(* IEC 61131-3 sources: plc_ladder_to_st/plc_export/st, 12 files *)

(* ---- P01_Main.st ---- *)
(* Generated ST from context: P01_Main *)
(* Project: plc project_260626 *)
(* CPU: QCPU (Q mode) Q06H *)

(* ============================================================ *)
(* [STEP 1] CODESYS > POU 열기 > DECLARATION(선언) 탭 > 아래만 붙여넣기 *)
(*          POU 이름과 PROGRAM 이름이 같아야 함: 'P01_Main' *)
(* ============================================================ *)

PROGRAM P01_Main
VAR
    SM400 : BOOL; (* 항상on *)
    M200 : BOOL; (* 제어전원ON *)
    X0 : BOOL; (* 운전준비ON [PBL] *)
    M201 : BOOL; (* 운전준비 PLS *)
    M202 : BOOL; (* 제어반 운전준비완료 *)
    M50 : BOOL; (* 제어반 비상정지 *)
    X1 : BOOL; (* 운전모드 자동[ ]  [SS] *)
    M210 : BOOL; (* 운전모드 수동[ ] *)
    M211 : BOOL; (* 운전모드 자동[ ] *)
    M500 : BOOL; (* 기동시작[HMI]   PB *)
    M215 : BOOL; (* 가와실러자동기동 *)
    M216 : BOOL; (* 현대 프라이머자동기동 *)
    M2127 : BOOL; (* 글라스 센터링 이상    TOTAL *)
    M2021 : BOOL; (* 글라스 센터링 운전준비 완료 *)
    X8 : BOOL; (* 이상해제[PB] *)
    M501 : BOOL; (* 이상해제[HMI]   PB *)
    M212 : BOOL; (* 이상해제 *)
    Y77 : BOOL; (* 선두 이더넷 카드 이상해제XY60 *)
    M502 : BOOL; (* 부저정지[HMI]   PB *)
    M220 : BOOL; (* 부져정지 SET *)
    M57 : BOOL; (* 설비 종합이상 *)
    X1100 : BOOL; (* 현대 작업완료    PRIMER] *)
    M170 : BOOL; (* 프라이머작업완료[HMI]   SET PB *)
    M171 : BOOL; (* 프라이머작업완료[HMI]   RST PB *)
    M710 : BOOL; (* 프라이머로보트[HMI]     PASS PB *)
    M1321 : BOOL; (* 프라이머로보트 작업완료 *)
    X111F : BOOL; (* 현대    PRIMER] HOME *)
    X1018 : BOOL; (* 실러 작업완료[ RB] *)
    M174 : BOOL; (* 실러작업완료[HMI] SET PB *)
    M175 : BOOL; (* 실러작업완료[HMI] RST PB *)
    M712 : BOOL; (* 실러 로보트[HMI]         PASS PB *)
    M60 : BOOL; (* 실러 로보트 작업완료 *)
    M2005 : BOOL; (* 센터링 글라스 감지단 *)
    M180 : BOOL; (* 글라스 반전 완료[HMI]      PB *)
    M2000 : BOOL; (* 센터링 가압 후진단 *)
    M2002 : BOOL; (* 센터링 이컬라이져 후진단 *)
    M1422 : BOOL; (* 센터링 글라스 로딩완료 *)
    M1522 : BOOL; (* 실러 센터링 완료 *)
    M5000 : BOOL; (* 실러비전OK *)
    M5001 : BOOL; (* 실러비전NG *)
    M6000 : BOOL; (* 바디비전OK *)
    M6001 : BOOL; (* 바디비전NG *)
    M6100 : BOOL; (* Gap Complete *)
    T70 : TON; (* 실러    ROBOT   HOME    POSITION *)
    M7750 : BOOL; (* Body    Auto    Start   COND *)
    M7000 : BOOL; (* 프라이머OK *)
    M7001 : BOOL; (* 프라이머NG *)
    T50 : TON; (* PRIMER  ROBOT   HOME    DELAY *)
    M7751 : BOOL; (* Primer  Auto    Start   COND *)
    X0_PLS : BOOL; (* 운전준비ON [PBL] *)
    X1018_PLS : BOOL; (* 실러 작업완료[ RB] *)
    X1100_PLS : BOOL; (* 현대 작업완료    PRIMER] *)
END_VAR

(* ============================================================ *)
(* [STEP 2] CODESYS > 같은 POU > IMPLEMENTATION(구현) 탭 > 아래만 붙여넣기 *)
(*          VAR 블록은 여기 넣으면 안 됨 *)
(* ============================================================ *)

(* --- Rung 1, step 0 | MODE --- *)
IF SM400 THEN
    M200 := TRUE;
ELSE
    M200 := FALSE;
END_IF;

(* --- Rung 2, step 6 --- *)
IF X0_PLS THEN
    M201 := TRUE;
ELSE
    M201 := FALSE;
END_IF;

(* --- Rung 3, step 8 --- *)
IF (((M201) AND (NOT (M202))) OR ((NOT (M201)) AND (M202))) AND (M200) AND (NOT (M50)) THEN
    M202 := TRUE;
ELSE
    M202 := FALSE;
END_IF;

(* --- Rung 4, step 16 --- *)
IF (M202) AND (NOT (X1)) THEN
    M210 := TRUE;
ELSE
    M210 := FALSE;
END_IF;

(* --- Rung 5, step 19 --- *)
IF (M202) AND (X1) THEN
    M211 := TRUE;
ELSE
    M211 := FALSE;
END_IF;

(* --- Rung 6, step 22 --- *)
IF ((M500) OR (M215)) AND (M211) AND (NOT (M50)) THEN
    M215 := TRUE;
ELSE
    M215 := FALSE;
END_IF;

(* --- Rung 7, step 27 --- *)
IF ((M500) OR (M216)) AND (M211) AND (NOT (M50)) THEN
    M216 := TRUE;
ELSE
    M216 := FALSE;
END_IF;

(* --- Rung 8, step 32 --- *)
IF (M202) AND (NOT (M2127)) THEN
    M2021 := TRUE;
ELSE
    M2021 := FALSE;
END_IF;

(* --- Rung 9, step 35 | Error Reset --- *)
IF (X8) OR (M501) THEN
    M212 := TRUE;
ELSE
    M212 := FALSE;
END_IF;

(* --- Rung 10, step 46 --- *)
IF M212 THEN
    Y77 := TRUE;
ELSE
    Y77 := FALSE;
END_IF;

(* --- Rung 11, step 48 --- *)
IF (SM400) AND (M502) THEN
    M220 := TRUE;
END_IF;
IF (SM400) AND (NOT (M57)) THEN
    M220 := FALSE;
END_IF;

(* --- Rung 12, step 55 | Work --- *)
IF (X1100_PLS) OR ((M210) AND (M170) AND (NOT (M171))) OR (M710) THEN
    M1321 := TRUE;
END_IF;

(* --- Rung 13, step 66 --- *)
IF (M210) AND (M171) AND (X111F) THEN
    M1321 := FALSE;
END_IF;

(* --- Rung 14, step 84 | - --- *)
IF (X1018_PLS) OR ((M210) AND (M174) AND (NOT (M175))) OR (M712) THEN
    M60 := TRUE;
END_IF;

(* --- Rung 15, step 80 --- *)
IF (M210) AND (M175) AND (NOT (M174)) THEN
    M60 := FALSE;
END_IF;

(* --- Rung 16, step 84 | - --- *)
IF (M2005) AND (M180) AND (M2005) AND (M2000) AND (M2002) THEN
    M1422 := TRUE;
END_IF;

(* --- Rung 17, step 93 --- *)
IF (M1522) OR (M2005) THEN
    M1422 := FALSE;
END_IF;

(* --- Rung 18, step 96 --- *)
IF (NOT (M60)) AND (NOT (M5000)) AND (NOT (M5001)) AND (NOT (M6000)) AND (NOT (M6001)) AND (NOT (M6100)) AND (T70) THEN
    M7750 := TRUE;
ELSE
    M7750 := FALSE;
END_IF;

(* --- Rung 19, step 104 --- *)
IF (NOT (M1321)) AND (NOT (M7000)) AND (NOT (M7001)) AND (T50) THEN
    M7751 := TRUE;
ELSE
    M7751 := FALSE;
END_IF;

(* ---- P02_Lamp.st ---- *)
(* Generated ST from context: P02_Lamp *)
(* Project: plc project_260626 *)
(* CPU: QCPU (Q mode) Q06H *)

(* ============================================================ *)
(* [STEP 1] CODESYS > POU 열기 > DECLARATION(선언) 탭 > 아래만 붙여넣기 *)
(*          POU 이름과 PROGRAM 이름이 같아야 함: 'P02_Lamp' *)
(* ============================================================ *)

PROGRAM P02_Lamp
VAR
    M202 : BOOL; (* 제어반 운전준비완료 *)
    SM412 : BOOL; (* 초 클럭1 *)
    M503 : BOOL; (* 램프 테스트[HMI]       PB *)
    Y20 : BOOL; (* 운전준비ON PBL  LAMP *)
    M57 : BOOL; (* 설비 종합이상 *)
    Y3C : BOOL; (* 제어반 타워램프 적색  [ ] *)
    M210 : BOOL; (* 운전모드 수동[ ] *)
    Y3D : BOOL; (* 제어반 타워램프 황색  [ ] *)
    M211 : BOOL; (* 운전모드 자동[ ] *)
    M215 : BOOL; (* 가와실러자동기동 *)
    M216 : BOOL; (* 현대 프라이머자동기동 *)
    Y3E : BOOL; (* 제어반 타워램프 녹색  [ ] *)
    M220 : BOOL; (* 부져정지 SET *)
    Y3F : BOOL; (* 제어반 타워램프 부져  [ ] *)
END_VAR

(* ============================================================ *)
(* [STEP 2] CODESYS > 같은 POU > IMPLEMENTATION(구현) 탭 > 아래만 붙여넣기 *)
(*          VAR 블록은 여기 넣으면 안 됨 *)
(* ============================================================ *)

(* --- Rung 1, step 0 --- *)
IF (M202) OR ((NOT (M202)) AND (SM412)) OR (M503) THEN
    Y20 := TRUE;
ELSE
    Y20 := FALSE;
END_IF;

(* --- Rung 2, step 6 --- *)
IF ((M57) AND (SM412)) OR (M503) THEN
    Y3C := TRUE;
ELSE
    Y3C := FALSE;
END_IF;

(* --- Rung 3, step 10 --- *)
IF ((M202) AND (M210)) OR (M503) THEN
    Y3D := TRUE;
ELSE
    Y3D := FALSE;
END_IF;

(* --- Rung 4, step 14 --- *)
IF ((M202) AND (((M211) AND (SM412)) OR ((M215) AND (M216)))) OR (M503) THEN
    Y3E := TRUE;
ELSE
    Y3E := FALSE;
END_IF;

(* --- Rung 5, step 23 --- *)
IF ((NOT (NOT (M57))) AND (NOT (M220))) OR (M503) THEN
    Y3F := TRUE;
ELSE
    Y3F := FALSE;
END_IF;

(* ---- P10_PrimerVision.st ---- *)
(* Generated ST from context: P10_PrimerVision *)
(* Project: plc project_260626 *)
(* CPU: QCPU (Q mode) Q06H *)

(* ============================================================ *)
(* [STEP 1] CODESYS > POU 열기 > DECLARATION(선언) 탭 > 아래만 붙여넣기 *)
(*          POU 이름과 PROGRAM 이름이 같아야 함: 'P10_PrimerVision' *)
(* ============================================================ *)

PROGRAM P10_PrimerVision
VAR
    SM401 : BOOL; (* 항상off *)
    D100 : WORD; (* 프라이머비전 → PLC *)
    T210 : TON; (* 프라이머비전 라이브 비트지연 *)
    SM400 : BOOL; (* 항상on *)
    T200 : TON; (* 프라이머비전 통신이상 *)
    SM412 : BOOL; (* 초 클럭1 *)
    D110 : WORD; (* 프라이머비전PLC → *)
    X1104 : BOOL; (* 현대 비전 스타트    PRIMER] *)
    M720 : BOOL;
    D110_0 : BOOL; (* 프라이머비전PLC → *)
    D110_1 : BOOL; (* 프라이머비전PLC → *)
    X1105 : BOOL; (* 현대 비전    PRIMER]  OFF *)
    M721 : BOOL;
    D110_2 : BOOL; (* 프라이머비전PLC → *)
    M1321 : BOOL; (* 프라이머로보트 작업완료 *)
    M722 : BOOL;
    M210 : BOOL; (* 운전모드 수동[ ] *)
    M171 : BOOL; (* 프라이머작업완료[HMI]   RST PB *)
    X111F : BOOL; (* 현대    PRIMER] HOME *)
    M723 : BOOL;
    X1106 : BOOL; (* 현대 포지션    PRIMER] _1 *)
    D110_8 : BOOL; (* 프라이머비전PLC → *)
    X1107 : BOOL; (* 현대 포지션    PRIMER] _2 *)
    D110_9 : BOOL; (* 프라이머비전PLC → *)
    X1108 : BOOL; (* 현대 포지션    PRIMER] _4 *)
    X1109 : BOOL; (* 현대 포지션    PRIMER] _8 *)
    D100_0 : BOOL; (* 프라이머비전 → PLC *)
    M7000 : BOOL; (* 프라이머OK *)
    D100_1 : BOOL; (* 프라이머비전 → PLC *)
    M7001 : BOOL; (* 프라이머NG *)
END_VAR

(* ============================================================ *)
(* [STEP 2] CODESYS > 같은 POU > IMPLEMENTATION(구현) 탭 > 아래만 붙여넣기 *)
(*          VAR 블록은 여기 넣으면 안 됨 *)
(* ============================================================ *)

(* --- Rung 1, step 0 | Live Bit --- *)
IF (SM401) AND (D100_F) AND (T210) THEN
    D100_F := FALSE;
END_IF;
IF (SM401) AND (D100_F) THEN
    T210(IN := TRUE, PT := T#500s);
ELSE
    T210(IN := FALSE);
END_IF;

(* --- Rung 2, step 16 --- *)
IF (SM400) AND (NOT (D100_F)) THEN
    T200(IN := TRUE, PT := T#10s);
ELSE
    T200(IN := FALSE);
END_IF;

(* --- Rung 3, step 22 --- *)
IF (SM400) AND (SM412) THEN
    D110_F := TRUE;
ELSE
    D110_F := FALSE;
END_IF;

(* --- Rung 4, step 25 | Vision Start --- *)
IF (X1104) OR (M720) THEN
    D110_0 := TRUE;
ELSE
    D110_0 := FALSE;
END_IF;

(* --- Rung 5, step 36 --- *)
IF (X1104) OR (M720) THEN
    D110_1 := TRUE;
ELSE
    D110_1 := FALSE;
END_IF;

(* --- Rung 6, step 39 --- *)
IF (X1105) OR (M721) THEN
    D110_2 := TRUE;
ELSE
    D110_2 := FALSE;
END_IF;

(* --- Rung 7, step 42 --- *)
IF (M1321) OR (M722) THEN
    D110_E := TRUE;
ELSE
    D110_E := FALSE;
END_IF;

(* --- Rung 8, step 45 --- *)
IF ((M210) AND (M171) AND (X111F)) OR (M723) THEN
    D110_C := TRUE;
ELSE
    D110_C := FALSE;
END_IF;

(* --- Rung 9, step 50 | POS --- *)
IF (SM400) AND (X1106) THEN
    D110_8 := TRUE;
ELSE
    D110_8 := FALSE;
END_IF;
IF (SM400) AND (X1107) THEN
    D110_9 := TRUE;
ELSE
    D110_9 := FALSE;
END_IF;
IF (SM400) AND (X1108) THEN
    D110_A := TRUE;
ELSE
    D110_A := FALSE;
END_IF;
IF (SM400) AND (X1109) THEN
    D110_B := TRUE;
ELSE
    D110_B := FALSE;
END_IF;

(* --- Rung 10, step 67 --- *)
IF D100_0 THEN
    M7000 := TRUE;
END_IF;

(* --- Rung 11, step 69 --- *)
IF (M210) AND (M171) AND (X111F) THEN
    M7000 := FALSE;
END_IF;

(* --- Rung 12, step 73 --- *)
IF D100_1 THEN
    M7001 := TRUE;
END_IF;

(* --- Rung 13, step 75 --- *)
IF (M210) AND (M171) AND (X111F) THEN
    M7001 := FALSE;
END_IF;

(* ---- P11_SealerVision.st ---- *)
(* Generated ST from context: P11_SealerVision *)
(* Project: plc project_260626 *)
(* CPU: QCPU (Q mode) Q06H *)

(* ============================================================ *)
(* [STEP 1] CODESYS > POU 열기 > DECLARATION(선언) 탭 > 아래만 붙여넣기 *)
(*          POU 이름과 PROGRAM 이름이 같아야 함: 'P11_SealerVision' *)
(* ============================================================ *)

PROGRAM P11_SealerVision
VAR
    SM400 : BOOL; (* 항상on *)
    D200 : WORD; (* 실러비전→ PLC *)
    T201 : TON; (* 실러비전통신이상 *)
    SM412 : BOOL; (* 초 클럭1 *)
    D210 : WORD; (* 실러비전PLC → *)
    X100B : BOOL; (* 실러 구간[ RB]  1 *)
    D210_8 : BOOL; (* 실러비전PLC → *)
    X100C : BOOL; (* 실러 구간[ RB]  2 *)
    D210_9 : BOOL; (* 실러비전PLC → *)
    X100D : BOOL; (* 실러 구간[ RB]  4 *)
    X100E : BOOL; (* 실러 구간[ RB]  8 *)
    X1009 : BOOL; (* 실러 실러비전스타트[ RB] *)
    D210_0 : BOOL; (* 실러비전PLC → *)
    D210_1 : BOOL; (* 실러비전PLC → *)
    X100A : BOOL; (* 실러 실러비전[ RB] OFF *)
    D210_2 : BOOL; (* 실러비전PLC → *)
    M60 : BOOL; (* 실러 로보트 작업완료 *)
    M210 : BOOL; (* 운전모드 수동[ ] *)
    M175 : BOOL; (* 실러작업완료[HMI] RST PB *)
    M174 : BOOL; (* 실러작업완료[HMI] SET PB *)
    D200_0 : BOOL; (* 실러비전→ PLC *)
    M5000 : BOOL; (* 실러비전OK *)
    D200_1 : BOOL; (* 실러비전→ PLC *)
    M5001 : BOOL; (* 실러비전NG *)
END_VAR

(* ============================================================ *)
(* [STEP 2] CODESYS > 같은 POU > IMPLEMENTATION(구현) 탭 > 아래만 붙여넣기 *)
(*          VAR 블록은 여기 넣으면 안 됨 *)
(* ============================================================ *)

(* --- Rung 1, step 0 --- *)
IF (SM400) AND (D200_F) THEN
    T201(IN := TRUE, PT := T#5s);
ELSE
    T201(IN := FALSE);
END_IF;
IF (SM400) AND (SM412) THEN
    D210_F := TRUE;
ELSE
    D210_F := FALSE;
END_IF;

(* --- Rung 2, step 10 | POS --- *)
IF (SM400) AND (X100B) THEN
    D210_8 := TRUE;
ELSE
    D210_8 := FALSE;
END_IF;
IF (SM400) AND (X100C) THEN
    D210_9 := TRUE;
ELSE
    D210_9 := FALSE;
END_IF;
IF (SM400) AND (X100D) THEN
    D210_A := TRUE;
ELSE
    D210_A := FALSE;
END_IF;
IF (SM400) AND (X100E) THEN
    D210_B := TRUE;
ELSE
    D210_B := FALSE;
END_IF;

(* --- Rung 3, step 27 --- *)
IF X1009 THEN
    D210_0 := TRUE;
ELSE
    D210_0 := FALSE;
END_IF;

(* --- Rung 4, step 29 --- *)
IF X1009 THEN
    D210_1 := TRUE;
ELSE
    D210_1 := FALSE;
END_IF;

(* --- Rung 5, step 31 --- *)
IF X100A THEN
    D210_2 := TRUE;
ELSE
    D210_2 := FALSE;
END_IF;

(* --- Rung 6, step 33 --- *)
IF M60 THEN
    D210_E := TRUE;
ELSE
    D210_E := FALSE;
END_IF;

(* --- Rung 7, step 35 --- *)
IF (M210) AND (M175) AND (NOT (M174)) THEN
    D210_C := TRUE;
ELSE
    D210_C := FALSE;
END_IF;

(* --- Rung 8, step 39 --- *)
IF D200_0 THEN
    M5000 := TRUE;
END_IF;

(* --- Rung 9, step 41 --- *)
IF (M210) AND (M175) AND (NOT (M174)) THEN
    M5000 := FALSE;
END_IF;

(* --- Rung 10, step 45 --- *)
IF D200_1 THEN
    M5001 := TRUE;
END_IF;

(* --- Rung 11, step 47 --- *)
IF (M210) AND (M175) AND (NOT (M174)) THEN
    M5001 := FALSE;
END_IF;

(* ---- P12_BodyVision.st ---- *)
(* Generated ST from context: P12_BodyVision *)
(* Project: plc project_260626 *)
(* CPU: QCPU (Q mode) Q06H *)

(* ============================================================ *)
(* [STEP 1] CODESYS > POU 열기 > DECLARATION(선언) 탭 > 아래만 붙여넣기 *)
(*          POU 이름과 PROGRAM 이름이 같아야 함: 'P12_BodyVision' *)
(* ============================================================ *)

PROGRAM P12_BodyVision
VAR
    X1011 : BOOL; (* 실러[ RB]BODY START *)
    D310_0 : BOOL;
    D310_1 : BOOL;
    X1012 : BOOL; (* 실러[ RB]GAP START *)
    D310_7 : BOOL;
    M60 : BOOL; (* 실러 로보트 작업완료 *)
    D310 : WORD;
    M210 : BOOL; (* 운전모드 수동[ ] *)
    M175 : BOOL; (* 실러작업완료[HMI] RST PB *)
    M174 : BOOL; (* 실러작업완료[HMI] SET PB *)
    D300_0 : BOOL;
    M6000 : BOOL; (* 바디비전OK *)
    D300_1 : BOOL;
    M6001 : BOOL; (* 바디비전NG *)
    D300_2 : BOOL;
    D300_3 : BOOL;
    M6100 : BOOL; (* Gap Complete *)
END_VAR

(* ============================================================ *)
(* [STEP 2] CODESYS > 같은 POU > IMPLEMENTATION(구현) 탭 > 아래만 붙여넣기 *)
(*          VAR 블록은 여기 넣으면 안 됨 *)
(* ============================================================ *)

(* --- Rung 1, step 0 --- *)
IF X1011 THEN
    D310_0 := TRUE;
ELSE
    D310_0 := FALSE;
END_IF;
IF X1011 THEN
    D310_1 := TRUE;
ELSE
    D310_1 := FALSE;
END_IF;

(* --- Rung 2, step 3 --- *)
IF X1012 THEN
    D310_7 := TRUE;
ELSE
    D310_7 := FALSE;
END_IF;

(* --- Rung 3, step 5 --- *)
IF M60 THEN
    D310_E := TRUE;
ELSE
    D310_E := FALSE;
END_IF;

(* --- Rung 4, step 7 --- *)
IF (M210) AND (M175) AND (NOT (M174)) THEN
    D310_C := TRUE;
ELSE
    D310_C := FALSE;
END_IF;

(* --- Rung 5, step 11 --- *)
IF D300_0 THEN
    M6000 := TRUE;
END_IF;

(* --- Rung 6, step 13 --- *)
IF (M210) AND (M175) AND (NOT (M174)) THEN
    M6000 := FALSE;
END_IF;

(* --- Rung 7, step 17 --- *)
IF D300_1 THEN
    M6001 := TRUE;
END_IF;

(* --- Rung 8, step 19 --- *)
IF (M210) AND (M175) AND (NOT (M174)) THEN
    M6001 := FALSE;
END_IF;

(* --- Rung 9, step 23 --- *)
IF (D300_2) OR (D300_3) THEN
    M6100 := TRUE;
END_IF;

(* --- Rung 10, step 26 --- *)
IF (M210) AND (M175) AND (NOT (M174)) THEN
    M6100 := FALSE;
END_IF;

(* ---- P20_PrimerRobot.st ---- *)
(* Generated ST from context: P20_PrimerRobot *)
(* Project: plc project_260626 *)
(* CPU: QCPU (Q mode) Q06H *)

(* ============================================================ *)
(* [STEP 1] CODESYS > POU 열기 > DECLARATION(선언) 탭 > 아래만 붙여넣기 *)
(*          POU 이름과 PROGRAM 이름이 같아야 함: 'P20_PrimerRobot' *)
(* ============================================================ *)

PROGRAM P20_PrimerRobot
VAR
    X111F : BOOL; (* 현대    PRIMER] HOME *)
    T50 : TON; (* PRIMER  ROBOT   HOME    DELAY *)
    M1353 : BOOL; (* PRIMER  ROBOT   HOME    (M1350.3 *)
    M1321 : BOOL; (* 프라이머로보트 작업완료 *)
    M50 : BOOL; (* 제어반 비상정지 *)
    M7751 : BOOL; (* Primer  Auto    Start   COND *)
    M1362 : BOOL; (* PRIMER  RB STARTCONDITION *)
    X7 : BOOL; (* 로보트 재기동    [PB] *)
    X1119 : BOOL; (* 현대[    PRIMER] program end *)
    M1364 : BOOL; (* 로봇 재기동PRIMER        (M1352.2 *)
    M216 : BOOL; (* 현대 프라이머자동기동 *)
    X111D : BOOL; (* 현대 로봇    PRIMER] Auto mode *)
    X111E : BOOL; (* 현대    PRIMER] Robot   Ready On *)
    X111A : BOOL; (* 현대    PRIMER] Robot   Error *)
    M710 : BOOL; (* 프라이머로보트[HMI]     PASS PB *)
    T51 : TON; (* PRIMER  ROBOT   START   DELAY *)
    T52 : TON; (* PRIMER  ROBOT   START   OFF *)
    X111C : BOOL; (* 현대    PRIMER] Robot   Running *)
    Y1116 : BOOL; (* 현대    PRIMER] ROBOT   START *)
    X1117 : BOOL; (* 현대 로봇 비상정지    PRIMER] *)
    X1036 : BOOL; (* 실러 로보트 비상정지[ RB] *)
    Y1117 : BOOL; (* 현대    PRIMER] ROBOT   PAUSE *)
    M212 : BOOL; (* 이상해제 *)
    Y1103 : BOOL; (* 현대 로봇 이상해제    PRIMER] *)
    X1101 : BOOL; (* 현대 센터링 간섭무    PRIMER] *)
    M1354 : BOOL; (* 불간섭PRIMER  ROBOT     (M1350.4 *)
    SM400 : BOOL; (* 항상on *)
    Y1100 : BOOL; (* 현대 센터링 진입가능    PRIMER] *)
    X1002 : BOOL; (* 실러 프라이머로봇 상호인터록[ RB] *)
    M712 : BOOL; (* 실러 로보트[HMI]         PASS PB *)
    X103D : BOOL; (* 실러[ RB]HOME    POSITION *)
    Y1102 : BOOL; (* 현대 실러 상호인터록    PRIMER] RB *)
    M700 : BOOL; (* 프라이머로보트 선택  _HMIPB *)
    M701 : BOOL; (* 비젼 로보트 선택      _HMIPB *)
    M702 : BOOL; (* 실러 로보트 선택      _HMIPB *)
    M600 : BOOL; (* 프라이머차종선택1 HMI *)
    M601 : BOOL; (* 프라이머차종선택2 HMI *)
    M602 : BOOL; (* 프라이머차종선택4 HMI *)
    D600 : WORD; (* 프라이머차종입력 *)
    D700 : WORD; (* 프라이머차종 *)
    X111F_PLS : BOOL; (* 현대    PRIMER] HOME *)
END_VAR

(* ============================================================ *)
(* [STEP 2] CODESYS > 같은 POU > IMPLEMENTATION(구현) 탭 > 아래만 붙여넣기 *)
(*          VAR 블록은 여기 넣으면 안 됨 *)
(* ============================================================ *)

(* --- Rung 1, step 0 | HOME --- *)
IF (X111F) AND (T50) THEN
    M1353 := TRUE;
ELSE
    M1353 := FALSE;
END_IF;
IF X111F THEN
    T50(IN := TRUE, PT := T#1s);
ELSE
    T50(IN := FALSE);
END_IF;

(* --- Rung 2, step 13 | START --- *)
IF ((K0 <> K0)) AND (NOT (M1321)) AND (NOT (M50)) AND (M7751) THEN
    M1362 := TRUE;
ELSE
    M1362 := FALSE;
END_IF;

(* --- Rung 3, step 25 --- *)
IF (X7) AND ((NOT (X111F)) OR (X1119)) THEN
    M1364 := TRUE;
ELSE
    M1364 := FALSE;
END_IF;

(* --- Rung 4, step 30 --- *)
IF (M216) AND (((M1362) AND (T50)) OR ((M1364) AND (NOT (T50)))) AND (X111D) AND (X111E) AND (NOT (X111A)) AND (NOT (M710)) AND (T51) AND (NOT (T52)) AND (NOT (X111C)) AND (NOT (M710)) THEN
    Y1116 := TRUE;
ELSE
    Y1116 := FALSE;
END_IF;
IF (M216) AND (((M1362) AND (T50)) OR ((M1364) AND (NOT (T50)))) AND (X111D) AND (X111E) AND (NOT (X111A)) AND (NOT (M710)) THEN
    T51(IN := TRUE, PT := T#500ms);
ELSE
    T51(IN := FALSE);
END_IF;
IF (M216) AND (((M1362) AND (T50)) OR ((M1364) AND (NOT (T50)))) AND (X111D) AND (X111E) AND (NOT (X111A)) AND (NOT (M710)) THEN
    T52(IN := TRUE, PT := T#2s);
ELSE
    T52(IN := FALSE);
END_IF;

(* --- Rung 5, step 56 --- *)
IF (M216) AND (NOT (X1117)) AND (NOT (X1036)) THEN
    Y1117 := TRUE;
ELSE
    Y1117 := FALSE;
END_IF;

(* --- Rung 6, step 60 --- *)
IF M212 THEN
    Y1103 := TRUE;
ELSE
    Y1103 := FALSE;
END_IF;

(* --- Rung 7, step 62 | INPUT --- *)
IF (X1101) OR (M710) THEN
    M1354 := TRUE;
ELSE
    M1354 := FALSE;
END_IF;

(* --- Rung 8, step 70 | OUTPUT --- *)
IF SM400 THEN
    Y1100 := TRUE;
ELSE
    Y1100 := FALSE;
END_IF;

(* --- Rung 9, step 77 --- *)
IF (X1002) OR ((M712) AND (X103D)) THEN
    Y1102 := TRUE;
ELSE
    Y1102 := FALSE;
END_IF;

(* --- Rung 10, step 82 | Car Type --- *)
IF (SM400) AND (M700) AND (NOT (M701)) AND (NOT (M702)) AND (M600) THEN
    D700 := K1;
END_IF;
IF (SM400) AND (M700) AND (NOT (M701)) AND (NOT (M702)) AND (M601) THEN
    D700 := K2;
END_IF;
IF (SM400) AND (M700) AND (NOT (M701)) AND (NOT (M702)) AND (M602) THEN
    D700 := K3;
END_IF;
IF (SM400) AND (M700) AND (NOT (M701)) AND (NOT (M702)) THEN
    D700 := D600;
END_IF;
IF (SM400) AND (M700) AND (NOT (M701)) AND (NOT (M702)) THEN
    K1Y1118 := D700;
END_IF;

(* --- Rung 11, step 110 --- *)
IF X111F_PLS THEN
    D700 := K0;
END_IF;
IF X111F_PLS THEN
    D600 := K0;
END_IF;

(* ---- P21_BodyRobot.st ---- *)
(* Generated ST from context: P21_BodyRobot *)
(* Project: plc project_260626 *)
(* CPU: QCPU (Q mode) Q06H *)

(* ============================================================ *)
(* [STEP 1] CODESYS > POU 열기 > DECLARATION(선언) 탭 > 아래만 붙여넣기 *)
(*          POU 이름과 PROGRAM 이름이 같아야 함: 'P21_BodyRobot' *)
(* ============================================================ *)

PROGRAM P21_BodyRobot
VAR
    X103D : BOOL; (* 실러[ RB]HOME    POSITION *)
    T70 : TON; (* 실러    ROBOT   HOME    POSITION *)
    M1553 : BOOL; (* 실러    ROBOT   HOME    POSITION *)
    M1556 : BOOL; (* 실러로봇센터링 진입가능 반전  ( ) *)
    M2005 : BOOL; (* 센터링 글라스 감지단 *)
    M1522 : BOOL; (* 실러 센터링 완료 *)
    M50 : BOOL; (* 제어반 비상정지 *)
    M7750 : BOOL; (* Body    Auto    Start   COND *)
    M1552 : BOOL; (* 실러로봇START   CONDITION *)
    X7 : BOOL; (* 로보트 재기동    [PB] *)
    M1555 : BOOL; (* 실러 로봇재기동   (M1552.2 *)
    M215 : BOOL; (* 가와실러자동기동 *)
    X103C : BOOL; (* 실러[ RB]TEACH   MODE *)
    X103E : BOOL; (* 실러[ RB]MOTOR   POWER ON *)
    X103B : BOOL; (* 실러[ RB]ERROR *)
    M712 : BOOL; (* 실러 로보트[HMI]         PASS PB *)
    T71 : TON; (* 실러[ RB]ROBOT   START   DELAY *)
    T72 : TON; (* 실러[ RB]ROBOT   START   OFF *)
    Y1030 : BOOL; (* 실러[ RB]external_cycle   start *)
    Y1032 : BOOL; (* 실러[ RB]RPS ON  (Q206.2) *)
    Y1035 : BOOL; (* 실러[ RB]MOTOR ON *)
    X1117 : BOOL; (* 현대 로봇 비상정지    PRIMER] *)
    X1036 : BOOL; (* 실러 로보트 비상정지[ RB] *)
    Y1033 : BOOL; (* 가와실러[ ]external hold *)
    M212 : BOOL; (* 이상해제 *)
    Y1034 : BOOL; (* 실러[ RB]external hold   RESET *)
    Y1031 : BOOL; (* 실러[ RB]external error  reset *)
    X1000 : BOOL; (* 실러 센터링 간섭무[ RB] *)
    M1554 : BOOL; (* 실러 간섭무    ROBOT *)
    M2003 : BOOL; (* 센터링 이컬라이져 전진단 *)
    M2001 : BOOL; (* 센터링 가압 전진단 *)
    X1007 : BOOL; (* 실러 센터링 언클램프요구[ RB] *)
    M1421 : BOOL; (* 센터링 언클램프 요구      (M1422.1 *)
    Y1000 : BOOL; (* 실러 센터링 진입가능[ RB] *)
    Y100A : BOOL; (* 실러 실러비젼[ RB]  NG *)
    Y100C : BOOL; (* 실러 바디비젼[ RB] NG *)
    M2000 : BOOL; (* 센터링 가압 후진단 *)
    M2002 : BOOL; (* 센터링 이컬라이져 후진단 *)
    Y1001 : BOOL; (* 실러 바디 진입[ RB]  OK *)
    Y48 : BOOL; (* 실링 카트리지정회전 토출      [ ] *)
    Y4C : BOOL; (* 컨트롤러속도선택DM300   1 *)
    X111F : BOOL; (* 현대    PRIMER] HOME *)
    M710 : BOOL; (* 프라이머로보트[HMI]     PASS PB *)
    X1A : BOOL; (* 실링 카트리지후진단 *)
    M999 : BOOL;
    Y1002 : BOOL; (* 실러 실러 진입[ RB]  OK *)
    M3000 : BOOL; (* 그리퍼 진공흡착확인 *)
    Y1003 : BOOL; (* 실러 진공흡착확인[ RB]  OK *)
    M3001 : BOOL; (* 그리퍼 진공탈착확인 *)
    Y1004 : BOOL; (* 실러 진공탈착확인[ RB]  OK *)
    Y1005 : BOOL; (* 실러 센터링 언클램프[ RB]   OK *)
    X1102 : BOOL; (* 현대 실러 상호인터록    PRIMER] RB *)
    Y1018 : BOOL; (* 실러 프라이머로봇 상호인터록[ RB] *)
    SM400 : BOOL; (* 항상on *)
    M5000 : BOOL; (* 실러비전OK *)
    M5001 : BOOL; (* 실러비전NG *)
    Y1009 : BOOL; (* 실러 실러비젼[ RB] OK *)
    M6000 : BOOL; (* 바디비전OK *)
    M6001 : BOOL; (* 바디비전NG *)
    Y100B : BOOL; (* 실러 바디비전[ RB] OK *)
    M6100 : BOOL; (* Gap Complete *)
    Y100D : BOOL; (* 실러[ RB]GAP COMP *)
    M181 : BOOL; (* PC      Change  Complete *)
    T700 : TON;
    Y100F : BOOL;
    M702 : BOOL; (* 실러 로보트 선택      _HMIPB *)
    M700 : BOOL; (* 프라이머로보트 선택  _HMIPB *)
    M701 : BOOL; (* 비젼 로보트 선택      _HMIPB *)
    M620 : BOOL; (* 실러 차종선택    1 HMI *)
    M621 : BOOL; (* 실러 차종선택   2 HMI *)
    M622 : BOOL; (* 실러 차종선택   4 *)
    D620 : WORD; (* 실러 차종입력 *)
    D720 : WORD; (* 실러차종 *)
    X103D_PLS : BOOL; (* 실러[ RB]HOME    POSITION *)
END_VAR

(* ============================================================ *)
(* [STEP 2] CODESYS > 같은 POU > IMPLEMENTATION(구현) 탭 > 아래만 붙여넣기 *)
(*          VAR 블록은 여기 넣으면 안 됨 *)
(* ============================================================ *)

(* --- Rung 1, step 0 | HOME --- *)
IF (X103D) AND (T70) THEN
    M1553 := TRUE;
ELSE
    M1553 := FALSE;
END_IF;
IF X103D THEN
    T70(IN := TRUE, PT := T#1s);
ELSE
    T70(IN := FALSE);
END_IF;

(* --- Rung 2, step 13 | START --- *)
IF ((K0 <> K0)) AND (M1556) AND (M2005) AND (M1522) AND (NOT (M50)) AND (M7750) THEN
    M1552 := TRUE;
ELSE
    M1552 := FALSE;
END_IF;

(* --- Rung 3, step 27 --- *)
IF (X7) AND (NOT (X103D)) THEN
    M1555 := TRUE;
ELSE
    M1555 := FALSE;
END_IF;

(* --- Rung 4, step 30 --- *)
IF (M215) AND (((M1552) AND (T70)) OR ((M1555) AND (NOT (T70)))) AND (NOT (X103C)) AND (X103E) AND (NOT (X103B)) AND (NOT (M712)) AND (T71) AND (NOT (T72)) AND (NOT (M712)) THEN
    Y1030 := TRUE;
ELSE
    Y1030 := FALSE;
END_IF;
IF (M215) AND (((M1552) AND (T70)) OR ((M1555) AND (NOT (T70)))) AND (NOT (X103C)) AND (X103E) AND (NOT (X103B)) AND (NOT (M712)) AND (T71) AND (NOT (T72)) AND (NOT (M712)) THEN
    Y1032 := TRUE;
ELSE
    Y1032 := FALSE;
END_IF;
IF (M215) AND (((M1552) AND (T70)) OR ((M1555) AND (NOT (T70)))) AND (NOT (X103C)) AND (X103E) AND (NOT (X103B)) AND (NOT (M712)) THEN
    T71(IN := TRUE, PT := T#500ms);
ELSE
    T71(IN := FALSE);
END_IF;
IF (M215) AND (((M1552) AND (T70)) OR ((M1555) AND (NOT (T70)))) AND (NOT (X103C)) AND (X103E) AND (NOT (X103B)) AND (NOT (M712)) THEN
    T72(IN := TRUE, PT := T#2s);
ELSE
    T72(IN := FALSE);
END_IF;

(* --- Rung 5, step 56 --- *)
IF (M215) AND (NOT (X103E)) THEN
    Y1035 := TRUE;
ELSE
    Y1035 := FALSE;
END_IF;

(* --- Rung 6, step 59 --- *)
IF (M215) AND (NOT (X1117)) AND (NOT (X1036)) THEN
    Y1033 := TRUE;
ELSE
    Y1033 := FALSE;
END_IF;

(* --- Rung 7, step 63 --- *)
IF (M212) OR (Y1030) THEN
    Y1034 := TRUE;
ELSE
    Y1034 := FALSE;
END_IF;

(* --- Rung 8, step 66 --- *)
IF M212 THEN
    Y1031 := TRUE;
ELSE
    Y1031 := FALSE;
END_IF;

(* --- Rung 9, step 68 | INPUT --- *)
IF X1000 THEN
    M1554 := TRUE;
ELSE
    M1554 := FALSE;
END_IF;

(* --- Rung 10, step 75 --- *)
IF (M215) AND ((M2003) OR (M2001)) AND (X1007) THEN
    M1421 := TRUE;
ELSE
    M1421 := FALSE;
END_IF;

(* --- Rung 11, step 81 | OUTPUT --- *)
IF (M215) AND (M1522) AND (M2005) THEN
    M1556 := TRUE;
ELSE
    M1556 := FALSE;
END_IF;

(* --- Rung 12, step 90 --- *)
IF M1556 THEN
    Y1000 := TRUE;
ELSE
    Y1000 := FALSE;
END_IF;

(* --- Rung 13, step 92 --- *)
IF ((Y100A) OR (Y100C)) AND (NOT (M2005)) AND (M2000) AND (M2002) THEN
    Y1001 := TRUE;
ELSE
    Y1001 := FALSE;
END_IF;

(* --- Rung 14, step 98 --- *)
IF (NOT (Y48)) AND (NOT (Y4C)) AND ((X111F) OR (M710)) AND ((X1A) OR (M999)) THEN
    Y1002 := TRUE;
ELSE
    Y1002 := FALSE;
END_IF;

(* --- Rung 15, step 107 --- *)
IF M3000 THEN
    Y1003 := TRUE;
ELSE
    Y1003 := FALSE;
END_IF;

(* --- Rung 16, step 109 --- *)
IF M3001 THEN
    Y1004 := TRUE;
ELSE
    Y1004 := FALSE;
END_IF;

(* --- Rung 17, step 111 --- *)
IF (M2000) AND (M2002) THEN
    Y1005 := TRUE;
ELSE
    Y1005 := FALSE;
END_IF;

(* --- Rung 18, step 114 --- *)
IF (X1102) OR ((M710) AND (M999)) THEN
    Y1018 := TRUE;
ELSE
    Y1018 := FALSE;
END_IF;

(* --- Rung 19, step 119 --- *)
IF (SM400) AND (M5000) AND (NOT (M5001)) THEN
    Y1009 := TRUE;
ELSE
    Y1009 := FALSE;
END_IF;
IF (SM400) AND (NOT (M5000)) AND (M5001) THEN
    Y100A := TRUE;
ELSE
    Y100A := FALSE;
END_IF;

(* --- Rung 20, step 128 --- *)
IF (SM400) AND (M6000) AND (NOT (M6001)) THEN
    Y100B := TRUE;
ELSE
    Y100B := FALSE;
END_IF;
IF (SM400) AND (NOT (M6000)) AND (M6001) THEN
    Y100C := TRUE;
ELSE
    Y100C := FALSE;
END_IF;

(* --- Rung 21, step 137 --- *)
IF M6100 THEN
    Y100D := TRUE;
ELSE
    Y100D := FALSE;
END_IF;

(* --- Rung 22, step 139 --- *)
IF (M181) AND (T700) THEN
    Y100F := TRUE;
ELSE
    Y100F := FALSE;
END_IF;
IF M181 THEN
    T700(IN := TRUE, PT := T#1s);
ELSE
    T700(IN := FALSE);
END_IF;

(* --- Rung 23, step 148 | Car Type --- *)
IF (SM400) AND (M702) AND (NOT (M700)) AND (NOT (M701)) AND (M620) THEN
    D720 := K1;
END_IF;
IF (SM400) AND (M702) AND (NOT (M700)) AND (NOT (M701)) AND (M621) THEN
    D720 := K2;
END_IF;
IF (SM400) AND (M702) AND (NOT (M700)) AND (NOT (M701)) AND (M622) THEN
    D720 := K3;
END_IF;
IF (SM400) AND (M702) AND (NOT (M700)) AND (NOT (M701)) THEN
    D720 := D620;
END_IF;
IF (SM400) AND (M702) AND (NOT (M700)) AND (NOT (M701)) THEN
    K1Y1038 := D720;
END_IF;

(* --- Rung 24, step 176 --- *)
IF X103D_PLS THEN
    D720 := K0;
END_IF;
IF X103D_PLS THEN
    D620 := K0;
END_IF;

(* ---- P30_Centering.st ---- *)
(* Generated ST from context: P30_Centering *)
(* Project: plc project_260626 *)
(* CPU: QCPU (Q mode) Q06H *)

(* ============================================================ *)
(* [STEP 1] CODESYS > POU 열기 > DECLARATION(선언) 탭 > 아래만 붙여넣기 *)
(*          POU 이름과 PROGRAM 이름이 같아야 함: 'P30_Centering' *)
(* ============================================================ *)

PROGRAM P30_Centering
VAR
    SM400 : BOOL; (* 항상on *)
    X10 : BOOL; (* 센터링 가압 후진단 *)
    T20 : TON; (* 센터링 가압 후진단 지연 *)
    M2000 : BOOL; (* 센터링 가압 후진단 *)
    T21 : TON; (* 센터링 가압 전진단 지연 *)
    M2001 : BOOL; (* 센터링 가압 전진단 *)
    X11 : BOOL; (* 센터링 이컬라이져 후진단 *)
    T22 : TON; (* 센터링 이컬라이져 후진단 *)
    M2002 : BOOL; (* 센터링 이컬라이져 후진단 *)
    T23 : TON; (* 센터링 이컬라이져 전진단 *)
    M2003 : BOOL; (* 센터링 이컬라이져 전진단 *)
    X14 : BOOL; (* 글라스 센터링 글라스 감지단 *)
    T35 : TON; (* 센터링 글라스 감지단 *)
    M2005 : BOOL; (* 센터링 글라스 감지단 *)
    M1522 : BOOL; (* 실러 센터링 완료 *)
    M2020 : BOOL; (* 글라스 센터링    HOME POS. *)
    M2021 : BOOL; (* 글라스 센터링 운전준비 완료 *)
    M210 : BOOL; (* 운전모드 수동[ ] *)
    M516 : BOOL; (* 센타링 원점복귀[HMI]     PB *)
    M2027 : BOOL; (* 글라스 센터링 원점복귀보조 *)
    M215 : BOOL; (* 가와실러자동기동 *)
    M1421 : BOOL; (* 센터링 언클램프 요구      (M1422.1 *)
    M511 : BOOL; (* 가압단 후진[HMI]     PB *)
    Y40 : BOOL; (* 센터링 가압 전진    SOL *)
    Y41 : BOOL; (* 센터링 가압 후진   SOL *)
    M1422 : BOOL; (* 센터링 글라스 로딩완료 *)
    M510 : BOOL; (* 가압단 전진[HMI]     PB *)
    M1554 : BOOL; (* 실러 간섭무    ROBOT *)
    M513 : BOOL; (* 이컬러이져 후진[HMI]   PB *)
    Y43 : BOOL; (* 센터링 이컬라이져 전진         SOL *)
    Y42 : BOOL; (* 센터링 이컬라이져 후진         SOL *)
    M512 : BOOL; (* 이컬러이져 전진[HMI]   PB *)
END_VAR

(* ============================================================ *)
(* [STEP 2] CODESYS > 같은 POU > IMPLEMENTATION(구현) 탭 > 아래만 붙여넣기 *)
(*          VAR 블록은 여기 넣으면 안 됨 *)
(* ============================================================ *)

(* --- Rung 1, step 0 | Senser --- *)
IF (SM400) AND (X10) AND (T20) THEN
    M2000 := TRUE;
ELSE
    M2000 := FALSE;
END_IF;
IF (SM400) AND (X10) THEN
    T20(IN := TRUE, PT := T#1s);
ELSE
    T20(IN := FALSE);
END_IF;
IF (SM400) AND (NOT (X10)) AND (T21) THEN
    M2001 := TRUE;
ELSE
    M2001 := FALSE;
END_IF;
IF (SM400) AND (NOT (X10)) THEN
    T21(IN := TRUE, PT := T#1s);
ELSE
    T21(IN := FALSE);
END_IF;

(* --- Rung 2, step 26 --- *)
IF (SM400) AND (X11) AND (T22) THEN
    M2002 := TRUE;
ELSE
    M2002 := FALSE;
END_IF;
IF (SM400) AND (X11) THEN
    T22(IN := TRUE, PT := T#1s);
ELSE
    T22(IN := FALSE);
END_IF;
IF (SM400) AND (NOT (X11)) AND (T23) THEN
    M2003 := TRUE;
ELSE
    M2003 := FALSE;
END_IF;
IF (SM400) AND (NOT (X11)) THEN
    T23(IN := TRUE, PT := T#1s);
ELSE
    T23(IN := FALSE);
END_IF;
IF (SM400) AND (X14) AND (T35) THEN
    M2005 := TRUE;
ELSE
    M2005 := FALSE;
END_IF;
IF (SM400) AND (X14) THEN
    T35(IN := TRUE, PT := T#3s);
ELSE
    T35(IN := FALSE);
END_IF;

(* --- Rung 3, step 57 --- *)
IF (M2001) AND (M2003) THEN
    M1522 := TRUE;
ELSE
    M1522 := FALSE;
END_IF;

(* --- Rung 4, step 60 --- *)
IF (M2000) AND (M2002) THEN
    M2020 := TRUE;
ELSE
    M2020 := FALSE;
END_IF;

(* --- Rung 5, step 63 | Home Return --- *)
IF (M2021) AND (M210) AND ((M516) OR (M2027)) AND (NOT (M2020)) THEN
    M2027 := TRUE;
ELSE
    M2027 := FALSE;
END_IF;

(* --- Rung 6, step 107 | - --- *)
IF (M2021) AND (((M215) AND (M1421)) OR ((M210) AND ((M511) OR (M2027)))) AND (M2002) AND (NOT (M2000)) AND (NOT (Y40)) THEN
    Y41 := TRUE;
ELSE
    Y41 := FALSE;
END_IF;

(* --- Rung 7, step 94 --- *)
IF (M2021) AND (((M215) AND (M2005) AND (M1422)) OR ((M210) AND (M510))) AND (M2002) AND (NOT (M2001)) AND (M1554) AND (NOT (Y41)) THEN
    Y40 := TRUE;
ELSE
    Y40 := FALSE;
END_IF;

(* --- Rung 8, step 107 | - --- *)
IF (M2021) AND (((M215) AND (M1421)) OR ((M210) AND ((M513) OR (M2027)))) AND (M2001) AND (NOT (M2002)) AND (NOT (Y43)) THEN
    Y42 := TRUE;
ELSE
    Y42 := FALSE;
END_IF;

(* --- Rung 9, step 123 --- *)
IF (M2021) AND (((M215) AND (M2005) AND (M1422)) OR ((M210) AND (M512))) AND (M2001) AND (NOT (M2003)) AND (M1554) AND (NOT (Y42)) THEN
    Y43 := TRUE;
ELSE
    Y43 := FALSE;
END_IF;

(* ---- P31_Sealer.st ---- *)
(* Generated ST from context: P31_Sealer *)
(* Project: plc project_260626 *)
(* CPU: QCPU (Q mode) Q06H *)

(* ============================================================ *)
(* [STEP 1] CODESYS > POU 열기 > DECLARATION(선언) 탭 > 아래만 붙여넣기 *)
(*          POU 이름과 PROGRAM 이름이 같아야 함: 'P31_Sealer' *)
(* ============================================================ *)

PROGRAM P31_Sealer
VAR
    SM400 : BOOL; (* 항상on *)
    X1A : BOOL; (* 실링 카트리지후진단 *)
    M2500 : BOOL; (* 실링 카트리지후진단 원점      [ ] *)
    X1B : BOOL; (* 실링 카트리지전진단 *)
    M2501 : BOOL; (* 실링 카트리지전진단 *)
    M2520 : BOOL; (* 실링 카트리지원점위치 *)
    M202 : BOOL; (* 제어반 운전준비완료 *)
    M2521 : BOOL; (* 실링 카트리지운전준비완료 *)
    M211 : BOOL; (* 운전모드 자동[ ] *)
    X1039 : BOOL; (* 실러[ RB]CYCLE   START *)
    M999 : BOOL;
    X1004 : BOOL; (* 실러 실러 토출[ RB]  ON *)
    M210 : BOOL; (* 운전모드 수동[ ] *)
    M522 : BOOL; (* 실링카트리지정회전[HMI] *)
    M523 : BOOL; (* 실링카트리지역회전[HMI] *)
    M521 : BOOL; (* 실러토출미사용[HMI]   PB *)
    Y49 : BOOL; (* 실링 카트리지역회전 원점      [ ] *)
    Y48 : BOOL; (* 실링 카트리지정회전 토출      [ ] *)
    M2527 : BOOL; (* 실링 카트리지원점복귀보조 *)
    M526 : BOOL; (* 실링 카트리지 원점복귀[HMI]    PB *)
    Y2B : BOOL; (* 실링 카트리지모터 브레이크 *)
    Y4C : BOOL; (* 컨트롤러속도선택DM300   1 *)
    Y4A : BOOL; (* 실링 모터 알람해제속도선택  2 *)
END_VAR

(* ============================================================ *)
(* [STEP 2] CODESYS > 같은 POU > IMPLEMENTATION(구현) 탭 > 아래만 붙여넣기 *)
(*          VAR 블록은 여기 넣으면 안 됨 *)
(* ============================================================ *)

(* --- Rung 1, step 0 --- *)
IF (SM400) AND (X1A) THEN
    M2500 := TRUE;
ELSE
    M2500 := FALSE;
END_IF;
IF (SM400) AND (X1B) THEN
    M2501 := TRUE;
ELSE
    M2501 := FALSE;
END_IF;

(* --- Rung 2, step 7 --- *)
IF (X1A) AND (NOT (X1B)) THEN
    M2520 := TRUE;
ELSE
    M2520 := FALSE;
END_IF;

(* --- Rung 3, step 10 --- *)
IF M202 THEN
    M2521 := TRUE;
ELSE
    M2521 := FALSE;
END_IF;

(* --- Rung 4, step 12 --- *)
IF (M2521) AND (((M211) AND ((X1039) OR (M999)) AND (X1004)) OR ((M210) AND ((M522) OR (X1004)) AND (NOT (M523)))) AND (NOT (M521)) AND (NOT (X1B)) AND (NOT (Y49)) THEN
    Y48 := TRUE;
ELSE
    Y48 := FALSE;
END_IF;

(* --- Rung 5, step 29 --- *)
IF (M2521) AND (((M211) AND (((X1B) AND (NOT (X1004))) OR (Y49))) OR ((M210) AND ((M523) OR (M2527)) AND (NOT (M522)))) AND ((NOT (M521)) OR (M999)) AND (NOT (X1A)) AND (NOT (Y48)) THEN
    Y49 := TRUE;
ELSE
    Y49 := FALSE;
END_IF;

(* --- Rung 6, step 48 --- *)
IF (M2521) AND (M210) AND ((M526) OR (M2527)) AND (NOT (X1A)) THEN
    M2527 := TRUE;
ELSE
    M2527 := FALSE;
END_IF;

(* --- Rung 7, step 55 --- *)
IF NOT ((NOT (Y48)) AND (NOT (Y49))) THEN
    Y2B := TRUE;
ELSE
    Y2B := FALSE;
END_IF;

(* --- Rung 8, step 59 --- *)
IF Y48 THEN
    Y4C := TRUE;
ELSE
    Y4C := FALSE;
END_IF;

(* --- Rung 9, step 61 --- *)
IF Y49 THEN
    Y4A := TRUE;
ELSE
    Y4A := FALSE;
END_IF;

(* ---- P32_Primer.st ---- *)
(* Generated ST from context: P32_Primer *)
(* Project: plc project_260626 *)
(* CPU: QCPU (Q mode) Q06H *)

(* ============================================================ *)
(* [STEP 1] CODESYS > POU 열기 > DECLARATION(선언) 탭 > 아래만 붙여넣기 *)
(*          POU 이름과 PROGRAM 이름이 같아야 함: 'P32_Primer' *)
(* ============================================================ *)

PROGRAM P32_Primer
VAR
    X2 : BOOL;
    T2 : TON;
    M110 : BOOL; (* OLD     PRIMER *)
    M111 : BOOL; (* NEW     PRIMER *)
    X3 : BOOL;
    T3 : TON;
    X1103 : BOOL; (* 현대 프라이머토출    PRIMER]  ON *)
    M102 : BOOL; (* OLD     PRIMER  ON *)
    M103 : BOOL; (* OLD     PRIMER  OFF *)
    M100 : BOOL; (* NEW     PRIMER  ON *)
    SM400 : BOOL; (* 항상on *)
    Y2D : BOOL; (* 프라이머토출 ON *)
    T10 : TON;
    Y2E : BOOL; (* 프라이머토출 OFF *)
END_VAR

(* ============================================================ *)
(* [STEP 2] CODESYS > 같은 POU > IMPLEMENTATION(구현) 탭 > 아래만 붙여넣기 *)
(*          VAR 블록은 여기 넣으면 안 됨 *)
(* ============================================================ *)

(* --- Rung 1, step 0 --- *)
IF (X2) AND (T2) THEN
    M110 := TRUE;
END_IF;
IF X2 THEN
    M111 := FALSE;
END_IF;
IF X2 THEN
    T2(IN := TRUE, PT := T#1s);
ELSE
    T2(IN := FALSE);
END_IF;

(* --- Rung 2, step 10 --- *)
IF (X3) AND (T3) THEN
    M111 := TRUE;
END_IF;
IF X3 THEN
    M110 := FALSE;
END_IF;
IF X3 THEN
    T3(IN := TRUE, PT := T#1s);
ELSE
    T3(IN := FALSE);
END_IF;

(* --- Rung 3, step 20 --- *)
IF (M110) AND (X1103) THEN
    M102 := TRUE;
ELSE
    M102 := FALSE;
END_IF;
IF (M110) AND (NOT (X1103)) THEN
    M103 := TRUE;
ELSE
    M103 := FALSE;
END_IF;

(* --- Rung 4, step 27 --- *)
IF (M111) AND (X1103) THEN
    M100 := TRUE;
ELSE
    M100 := FALSE;
END_IF;

(* --- Rung 5, step 30 --- *)
IF (SM400) AND ((M102) OR (M100)) THEN
    Y2D := TRUE;
ELSE
    Y2D := FALSE;
END_IF;
IF (SM400) AND ((M103) OR (M100)) AND ((NOT (T10)) OR (M100)) THEN
    Y2E := TRUE;
ELSE
    Y2E := FALSE;
END_IF;
IF (SM400) AND ((M103) OR (M100)) THEN
    T10(IN := TRUE, PT := T#500ms);
ELSE
    T10(IN := FALSE);
END_IF;

(* ---- P33_Gripper.st ---- *)
(* Generated ST from context: P33_Gripper *)
(* Project: plc project_260626 *)
(* CPU: QCPU (Q mode) Q06H *)

(* ============================================================ *)
(* [STEP 1] CODESYS > POU 열기 > DECLARATION(선언) 탭 > 아래만 붙여넣기 *)
(*          POU 이름과 PROGRAM 이름이 같아야 함: 'P33_Gripper' *)
(* ============================================================ *)

PROGRAM P33_Gripper
VAR
    SM400 : BOOL; (* 항상on *)
    Y54 : BOOL; (* 가와사키로보트 진공  ON  SOL_1 *)
    Y56 : BOOL; (* 가와사키로보트 진공  ON  SOL_2 *)
    X1C : BOOL; (* 로보트 그리퍼 진공확인    #1 *)
    X1D : BOOL; (* 로보트 그리퍼 진공확인    #2 *)
    T25 : TON; (* 그리퍼 진공흡착확인 지연 *)
    M3000 : BOOL; (* 그리퍼 진공흡착확인 *)
    T26 : TON; (* 그리퍼 진공탈착확인 지연 *)
    M3001 : BOOL; (* 그리퍼 진공탈착확인 *)
    M3020 : BOOL; (* 실러 로보트 원위치 *)
    M202 : BOOL; (* 제어반 운전준비완료 *)
    M3127 : BOOL; (* 그리퍼 이상  TOTAL *)
    M3021 : BOOL; (* 실러 로보트 운전전비완료 *)
    X1005 : BOOL; (* 실러 그리퍼 진공흡착[ RB] *)
    X1006 : BOOL; (* 실러 그리퍼 진공탈착[ RB] *)
    M630 : BOOL; (* 실러 로봇그리퍼 진공 보조    ON *)
    M631 : BOOL; (* 실러 로봇그리퍼 진공 보조    OFF *)
    X1013 : BOOL;
    X1014 : BOOL;
    M633 : BOOL; (* SEALER  ROVOT   PUSH    ADV *)
    M634 : BOOL; (* SEALER  ROBOT   PUSH    REV *)
    M210 : BOOL; (* 운전모드 수동[ ] *)
    M215 : BOOL; (* 가와실러자동기동 *)
    M530 : BOOL; (* 진공흡착[HMI]   PB *)
    M531 : BOOL; (* 진공탈착[HMI]   PB *)
    Y46 : BOOL; (* 가와사키로보트 진공파기  SOL_1 *)
    Y47 : BOOL; (* 가와사키로보트 진공파기  SOL_2 *)
    T209 : TON; (* 진공 파기 SOL ON  TIME *)
    Y55 : BOOL; (* 가와사키로보트 진공  OFF SOL_1 *)
    Y57 : BOOL; (* 가와사키로보트 진공  OFF SOL_2 *)
    M7500 : BOOL;
    Y4E : BOOL; (* PUSH    ADV *)
    M7501 : BOOL;
    Y4D : BOOL; (* PUSH    REV *)
END_VAR

(* ============================================================ *)
(* [STEP 2] CODESYS > 같은 POU > IMPLEMENTATION(구현) 탭 > 아래만 붙여넣기 *)
(*          VAR 블록은 여기 넣으면 안 됨 *)
(* ============================================================ *)

(* --- Rung 1, step 0 --- *)
IF (SM400) AND ((Y54) OR (Y56)) AND (X1C) AND (X1D) AND (T25) THEN
    M3000 := TRUE;
ELSE
    M3000 := FALSE;
END_IF;
IF (SM400) AND ((Y54) OR (Y56)) AND (X1C) AND (X1D) THEN
    T25(IN := TRUE, PT := T#1s);
ELSE
    T25(IN := FALSE);
END_IF;

(* --- Rung 2, step 14 --- *)
IF (SM400) AND (NOT (Y54)) AND (NOT (Y56)) AND (NOT (X1C)) AND (NOT (X1D)) AND (T26) THEN
    M3001 := TRUE;
ELSE
    M3001 := FALSE;
END_IF;
IF (SM400) AND (NOT (Y54)) AND (NOT (Y56)) AND (NOT (X1C)) AND (NOT (X1D)) THEN
    T26(IN := TRUE, PT := T#1s);
ELSE
    T26(IN := FALSE);
END_IF;

(* --- Rung 3, step 27 --- *)
IF SM400 THEN
    M3020 := TRUE;
ELSE
    M3020 := FALSE;
END_IF;

(* --- Rung 4, step 29 --- *)
IF (M202) AND (NOT (M3127)) THEN
    M3021 := TRUE;
ELSE
    M3021 := FALSE;
END_IF;

(* --- Rung 5, step 32 --- *)
IF (SM400) AND (X1005) AND (NOT (X1006)) THEN
    M630 := TRUE;
ELSE
    M630 := FALSE;
END_IF;
IF (SM400) AND (X1006) AND (NOT (X1005)) THEN
    M631 := TRUE;
ELSE
    M631 := FALSE;
END_IF;
IF (SM400) AND (X1013) AND (NOT (X1014)) THEN
    M633 := TRUE;
ELSE
    M633 := FALSE;
END_IF;
IF (SM400) AND (NOT (X1013)) AND (X1014) THEN
    M634 := TRUE;
ELSE
    M634 := FALSE;
END_IF;

(* --- Rung 6, step 49 --- *)
IF (SM400) AND (((M210) AND (NOT (M215)) AND ((M530) OR (M630))) OR ((M215) AND ((M630) OR (Y54) OR (Y56)) AND (NOT (M631)))) THEN
    Y54 := TRUE;
ELSE
    Y54 := FALSE;
END_IF;
IF (SM400) AND (((M210) AND (NOT (M215)) AND ((M530) OR (M630))) OR ((M215) AND ((M630) OR (Y54) OR (Y56)) AND (NOT (M631)))) THEN
    Y56 := TRUE;
ELSE
    Y56 := FALSE;
END_IF;
IF (SM400) AND (((M210) AND (NOT (M215)) AND ((M531) OR (M631))) OR ((M215) AND ((M631) OR (Y46) OR (Y47)) AND (NOT (M630)) AND (NOT (T209)))) THEN
    Y55 := TRUE;
ELSE
    Y55 := FALSE;
END_IF;
IF (SM400) AND (((M210) AND (NOT (M215)) AND ((M531) OR (M631))) OR ((M215) AND ((M631) OR (Y46) OR (Y47)) AND (NOT (M630)) AND (NOT (T209)))) THEN
    Y57 := TRUE;
ELSE
    Y57 := FALSE;
END_IF;
IF (SM400) AND (((M210) AND (NOT (M215)) AND ((M531) OR (M631))) OR ((M215) AND ((M631) OR (Y46) OR (Y47)) AND (NOT (M630)) AND (NOT (T209)))) THEN
    Y46 := TRUE;
ELSE
    Y46 := FALSE;
END_IF;
IF (SM400) AND (((M210) AND (NOT (M215)) AND ((M531) OR (M631))) OR ((M215) AND ((M631) OR (Y46) OR (Y47)) AND (NOT (M630)) AND (NOT (T209)))) THEN
    Y47 := TRUE;
ELSE
    Y47 := FALSE;
END_IF;
IF (SM400) AND ((Y46) OR (Y47)) THEN
    T209(IN := TRUE, PT := T#5s);
ELSE
    T209(IN := FALSE);
END_IF;
IF (SM400) AND (T209) THEN
    M531 := FALSE;
END_IF;
IF (SM400) AND (M215) THEN
    M530 := FALSE;
END_IF;
IF (SM400) AND (M215) THEN
    M531 := FALSE;
END_IF;

(* --- Rung 7, step 100 --- *)
IF (M633) OR (M7500) THEN
    Y4E := TRUE;
ELSE
    Y4E := FALSE;
END_IF;

(* --- Rung 8, step 103 --- *)
IF (M634) OR (M7501) THEN
    Y4D := TRUE;
ELSE
    Y4D := FALSE;
END_IF;

(* ---- P99_Error.st ---- *)
(* Generated ST from context: P99_Error *)
(* Project: plc project_260626 *)
(* CPU: QCPU (Q mode) Q06H *)

(* ============================================================ *)
(* [STEP 1] CODESYS > POU 열기 > DECLARATION(선언) 탭 > 아래만 붙여넣기 *)
(*          POU 이름과 PROGRAM 이름이 같아야 함: 'P99_Error' *)
(* ============================================================ *)

PROGRAM P99_Error
VAR
    M54 : BOOL; (* 비상정지TOTAL *)
    M2127 : BOOL; (* 글라스 센터링 이상    TOTAL *)
    M3127 : BOOL; (* 그리퍼 이상  TOTAL *)
    M57 : BOOL; (* 설비 종합이상 *)
    X1F : BOOL; (* 제어반 비상정지  [EPBL] *)
    M50 : BOOL; (* 제어반 비상정지 *)
    M212 : BOOL; (* 이상해제 *)
    SM401 : BOOL; (* 항상off *)
    M51 : BOOL; (* 프라이머로보트 비상정지 *)
    M52 : BOOL; (* 실러 로보트 비상정지 *)
    M53 : BOOL;
    Y40 : BOOL; (* 센터링 가압 전진    SOL *)
    M2000 : BOOL; (* 센터링 가압 후진단 *)
    Y41 : BOOL; (* 센터링 가압 후진   SOL *)
    M2001 : BOOL; (* 센터링 가압 전진단 *)
    T100 : TON; (* 글라스 센터링 가압단 이상      SOL *)
    M2100 : BOOL; (* 글라스 센터링 가압단 이상      SOL *)
    Y42 : BOOL; (* 센터링 이컬라이져 후진         SOL *)
    M2002 : BOOL; (* 센터링 이컬라이져 후진단 *)
    Y43 : BOOL; (* 센터링 이컬라이져 전진         SOL *)
    M2003 : BOOL; (* 센터링 이컬라이져 전진단 *)
    T101 : TON; (* 글라스센터링 이컬라이져 이상   SOL *)
    M2101 : BOOL; (* 글라스센터링 이컬라이져 이상   SOL *)
    Y54 : BOOL; (* 가와사키로보트 진공  ON  SOL_1 *)
    Y56 : BOOL; (* 가와사키로보트 진공  ON  SOL_2 *)
    X1C : BOOL; (* 로보트 그리퍼 진공확인    #1 *)
    X1D : BOOL; (* 로보트 그리퍼 진공확인    #2 *)
    M3100 : BOOL; (* 실러 로보트 그리퍼 진공이상 *)
    T110 : TON; (* 실러 로보트 그리퍼 진공이상 *)
END_VAR

(* ============================================================ *)
(* [STEP 2] CODESYS > 같은 POU > IMPLEMENTATION(구현) 탭 > 아래만 붙여넣기 *)
(*          VAR 블록은 여기 넣으면 안 됨 *)
(* ============================================================ *)

(* --- Rung 1, step 0 | Total Error --- *)
IF NOT ((NOT (M54)) AND (NOT (M2127)) AND (NOT (M3127))) THEN
    M57 := TRUE;
ELSE
    M57 := FALSE;
END_IF;

(* --- Rung 2, step 13 | MCP Error --- *)
IF (NOT (X1F)) OR ((M50) AND (NOT (M212))) THEN
    M50 := TRUE;
ELSE
    M50 := FALSE;
END_IF;

(* --- Rung 3, step 25 --- *)
IF (SM401) OR ((M51) AND (NOT (M212))) THEN
    M51 := TRUE;
ELSE
    M51 := FALSE;
END_IF;

(* --- Rung 4, step 30 --- *)
IF (SM401) OR ((M52) AND (NOT (M212))) THEN
    M52 := TRUE;
ELSE
    M52 := FALSE;
END_IF;

(* --- Rung 5, step 35 --- *)
IF NOT ((NOT (M50)) AND (NOT (M51)) AND (NOT (M52)) AND (NOT (M53))) THEN
    M54 := TRUE;
ELSE
    M54 := FALSE;
END_IF;

(* --- Rung 6, step 41 | Centering Error --- *)
IF ((((Y40) AND (NOT (M2000))) OR ((Y41) AND (NOT (M2001)))) AND (T100)) OR ((M2100) AND (NOT (M212))) THEN
    M2100 := TRUE;
ELSE
    M2100 := FALSE;
END_IF;
IF ((((Y40) AND (NOT (M2000))) OR ((Y41) AND (NOT (M2001)))) AND (T100)) OR ((M2100) AND (NOT (M212))) THEN
    T100(IN := TRUE, PT := T#8s);
ELSE
    T100(IN := FALSE);
END_IF;

(* --- Rung 7, step 65 --- *)
IF ((((Y42) AND (NOT (M2002))) OR ((Y43) AND (NOT (M2003)))) AND (T101)) OR ((M2101) AND (NOT (M212))) THEN
    M2101 := TRUE;
ELSE
    M2101 := FALSE;
END_IF;
IF ((((Y42) AND (NOT (M2002))) OR ((Y43) AND (NOT (M2003)))) AND (T101)) OR ((M2101) AND (NOT (M212))) THEN
    T101(IN := TRUE, PT := T#8s);
ELSE
    T101(IN := FALSE);
END_IF;

(* --- Rung 8, step 79 --- *)
IF NOT ((NOT (M2100)) AND (NOT (M2101))) THEN
    M2127 := TRUE;
ELSE
    M2127 := FALSE;
END_IF;

(* --- Rung 9, step 83 | Gripper Error --- *)
IF (((Y54) AND (Y56) AND ((NOT (X1C)) OR (X1D))) OR ((M3100) AND (NOT (M212)))) AND (T110) THEN
    M3100 := TRUE;
ELSE
    M3100 := FALSE;
END_IF;
IF ((Y54) AND (Y56) AND ((NOT (X1C)) OR (X1D))) OR ((M3100) AND (NOT (M212))) THEN
    T110(IN := TRUE, PT := T#3s);
ELSE
    T110(IN := FALSE);
END_IF;

(* --- Rung 10, step 108 --- *)
IF NOT (NOT (M3100)) THEN
    M3127 := TRUE;
ELSE
    M3127 := FALSE;
END_IF;
